{attribute 'qualified_only'}
TYPE E_TransportTube :
(
	BI1 := 0,
	BI5 := 1,
	BI8 := 2,
	BO4 := 3,
	BO5 := 4,
	BO6 := 5,
	BO9 := 6,
	BO10 := 7,
	BO12 := 8,
	BO13 := 9,
	BO14 := 10
) UINT;
END_TYPE

(* stored: Version 1.1.0.1, ProductVersion 3.1.4024.0
   DUT E_TransportTube: Id {26e13819-1baa-4350-8f0d-08839603bdb0} *)
